# EPICS autosave request: CARSApp/Db/XRM_fastmap.req
$(P)$(Q):basedir
$(P)$(Q):workdir
$(P)$(Q):filename
$(P)$(Q):format
$(P)$(Q):fileext
$(P)$(Q):scanfile
